// TIA Portal V17 export
// export: Created 2023-02-14T02:49:39.5432232Z, ExportSetting WithDefaults, DisplayName Totally Integrated Automation Portal, DisplayVersion V17, DisplayName TIA Portal Openness, DisplayVersion V17, DisplayName TIA Portal Teamcenter Gateway, DisplayVersion V17, DisplayName TIA Portal Version Control Interface, DisplayVersion V17, DisplayName SINAMICS Startdrive Advanced, DisplayVersion V17, DisplayName SINAMICS Startdrive G130, G150, S120, S150, SINAMICS MV, S210, DisplayVersion V17, DisplayName SINAMICS Startdrive G110M, G120, G120C, G120D, G120P, G115D, DisplayVersion V17, DisplayName STEP 7 Professional, DisplayVersion V17, DisplayName STEP 7 Safety, DisplayVersion V17, DisplayName WinCC Professional, DisplayVersion V17
FUNCTION_BLOCK "BFT_Tomato"   // FB365, LAD
{ S7_Optimized_Access := 'TRUE' }
VERSION : 0.1
// stored: AutoNumber false, IsIECCheckEnabled false, IsRetainMemResEnabled false, MemoryReserve 100, SetENOAutomatically false, UDAEnableTagReadback false
   VAR_INPUT
      IN_FBAV_Inload : Bool;
      IN_FBAV_Outlet : Bool;
      IN_FBAV_Transfer : Bool;
      IN_FBAV_CIP_Tank : Bool;
      IN_FBAV_CIP_Line : Bool;
      IN_FBAV_Vinegar : Bool;
      IN_FBAV_ProWater : Bool;
      IN_FBP_Inload : Bool;
      IN_FBP_Inload_SP : Real;
      IN_FBP_Transfer : Bool;
      IN_FBP_Transfer_SP : Real;
      IN_FBP_CIP : Bool;
      IN_FBP_CIP_Sp : Real;
      IN_LT01 : Real;
      "LCS Start" : Bool;
      "LCS Stop" : Bool;
      "LCS EMS" : Bool;
      IN_Dose_Run : Bool;
      IN_Dose_Held : Bool;
      IN_Dose_Complete : Bool;
      IN_Dose_Header_1 : Bool;
      IN_Dose_Header_2 : Bool;
      IN_Dose_Valve_Cmd : Bool;
      IN_Dose_Pump_Cmd : Bool;
      IN_Dose_Pump_Sp : Real;
      IN_Dose_LineOK : Bool;
      "Inload Busy" : Bool;
      "CIP Pulse" : Bool;
      "CIP Supply ON" : Bool;
      "CIP Req OK" : Bool;
      "CIP Complete" : Bool;
      "CIP Busy" : Bool;
      "Vinegar Available" : Bool;
      "Vinegar Tank Ready" : Bool;
      "Vinegar Prod Ready" : Bool;
      "Vinegar Valve Open" : Bool;
      "Vinegar Pump Run" : Bool;
      IN_FT_Vinegar : Real;
      ProWater_Req_OK : Bool;
      IN_LDT : Date_And_Time;
   END_VAR
   VAR_OUTPUT
      Out_AV_Inload : Bool;
      Out_AV_Outlet : Bool;
      Out_AV_Transfer : Bool;
      Out_AV_CIP_Tank : Bool;
      Out_AV_CIP_Line : Bool;
      Out_AV_Vinegar : Bool;
      Out_AV_ProWater : Bool;
      Out_P_Inload : Bool;
      Out_P_Inload_Sp : Real;
      Out_P_Transfer : Bool;
      Out_P_Transfer_Sp : Real;
      Out_P_CIP : Bool;
      Out_P_CIP_Sp : Real;
      Out_XA : Bool;
      Out_XA_Speed : Real;
      "Vinegar Req" : Bool;
      ProWater_Req : Bool;
      Out_CIP_Req : Bool;
      Out_CIP_LineOpen : Bool;
   END_VAR
   VAR
      Cmd : Struct
         Inload_Tomato : Bool;
         Inload_ProWater : Bool;
         Ready_for_Tranfer : Bool;
         CIP_Tank : Bool;
         CIP_Line : Bool;
         Agitator_SpeedMode : Bool;
         Agitator_Mode : Bool;
         Agitator_Man_OnOff : Bool;
      END_STRUCT;
   END_VAR
   VAR RETAIN
      Param : Struct
         SP_Level_LL : Real := 10.0;
         SP_Level_ML : Real := 80.0;
         SP_Level_HL : Real := 100.0;
         SP_Level_Agi_ON1 : Real := 20.0;
         SP_Level_Agi_OFF1 : Real := 60.0;
         SP_Level_Agi_ON2 : Real := 62.0;
         SP_Level_Agi_OFF2 : Real := 80.0;
         SP_Level_Agi_ON3 : Real := 82.0;
         Agitator_SP_Speed : Real := 50.0;
         SupplyPump_SP_Speed : Real := 80.0;
         L_Hi_Lim : Real := 100.0;
         L_Lo_Lim : Real := 0.0;
         L_Hys : Real := 2.0;
         FlushingTime : DInt := 10000;
         CIP_Trf_SP_Speed : Real := 80.0;
         CIP_Ret_ON_SP : Real := 5.0;
         CIP_Ret_OFF_SP : Real;
      END_STRUCT;
   END_VAR
   VAR
      State : Struct   // Tank in loading state
         Tank_LL : Bool;
         Tank_ML : Bool;
         Tank_HL : Bool;
         Tank_inCIP : Bool;
         Tank_CIP_Enable : Bool;
         Line_inCIP : Bool;
         Line_CIP_Enable : Bool;
         CIP_Return_On : Bool;
         Inloading : Bool;
         Inload_Enable : Bool;
         Ready_For_Transfer : Bool;
         Ready_For_Transfer_Ena : Bool;
         Tank_Available : Bool;
         Transfer_On_Prog : Bool;
         L_Agi_ON1 : Bool;
         L_Agi_ON2 : Bool;
         L_Agi_ON3 : Bool;
         "Dose EN" : Bool;
         Inloading_ProWater : Bool;
         Inloading_Tomato : Bool;
      END_STRUCT;
      Dose : Struct
         Dose_Start : DWord;
         Dose_Pause : DWord;
         Dose_Stop : DWord;
         Dose_State : DWord;
      END_STRUCT;
      alwaysON : Bool;
      L_Hys_Abs : Real;
      Hys_Level_HL : Real;
      Hys_Level_ML : Real;
      Hys_Level_LL : Real;
      Hys_Level_Agi : Real;
      r : Struct
         PosE1 : Bool;
         PosE2 : Bool;
         PosE3 : Bool;
         PosE4 : Bool;
         PosE5 : Bool;
         PosE6 : Bool;
         PosE7 : Bool;
         PosE8 : Bool;
         PosE9 : Bool;
         PosE10 : Bool;
         PosE11 : Bool;
         PosE12 : Bool;
         PosE13 : Bool;
         PosE14 : Bool;
         PosE15 : Bool;
         PosE16 : Bool;
         PosE17 : Bool;
         PosE18 : Bool;
         PosE19 : Bool;
         PosE20 : Bool;
         PosE21 : Bool;
         PosE22 : Bool;
         PosE23 : Bool;
         PosE24 : Bool;
         PosE25 : Bool;
         PosE26 : Bool;
         PosE27 : Bool;
         PosE28 : Bool;
         PosE29 : Bool;
         PosE30 : Bool;
         PosE31 : Bool;
         PosE32 : Bool;
      END_STRUCT;
      Actuator : Struct
         AV_Inload_Tomato : Bool;
         AV_Inload_ProWater : Bool;
         AV_Outlet : Bool;
         AV_Transfer : Bool;
         AV_CIP_Tank : Bool;
         AV_CIP_Line : Bool;
         P_Transfer : Bool;
         P_Inload : Bool;
         P_CIP : Bool;
         Agitator_level : Bool;
         LCS_OnOff : Bool;
      END_STRUCT;
      FlushingTim : TON_TIME;
      SPumpTim { S7_SetPoint := 'True'} : TON_TIME;
      AVinloadTim { S7_SetPoint := 'True'} : TON_TIME;
      L_AgiTim { S7_SetPoint := 'True'} : TON_TIME;
      SP_Vinegar { S7_SetPoint := 'True'} : "RawDose";
      Dose_Vinegar { S7_SetPoint := 'True'} : "DOSE";
      Vinegar_Ready_State { S7_SetPoint := 'True'} : Bool;
      Vinegar_EN : Bool;
      Pump_TF_On_Time { S7_SetPoint := 'True'} : TON_TIME;
   END_VAR
   VAR_TEMP   // added for the SCL form of the ladder/FBD networks
      _w1 : Bool;
      _w2 : Bool;
   END_VAR
BEGIN

REGION Network 1: Always_ON
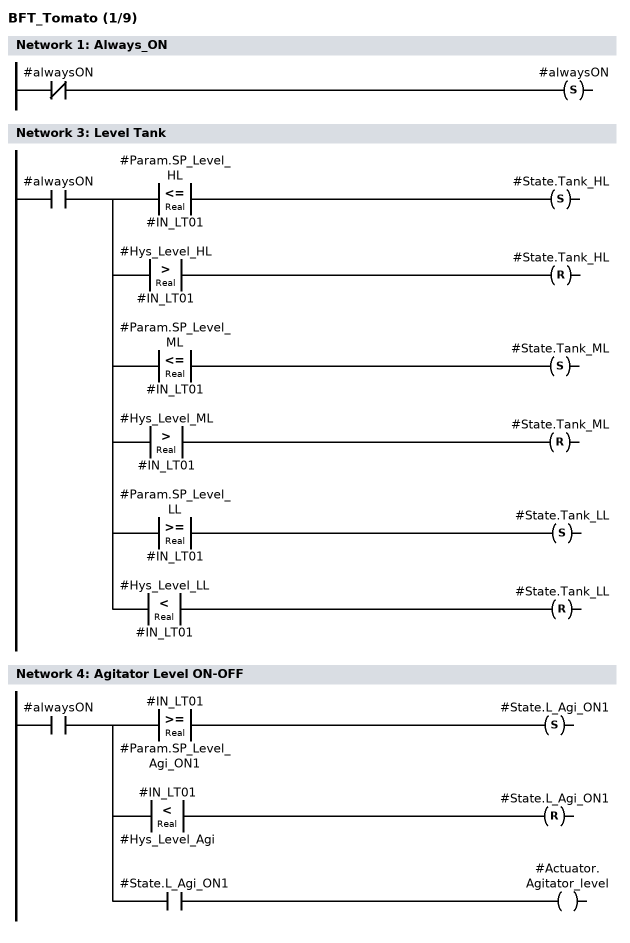
   RUNG wire#powerrail
      I_Contact( #alwaysON )
      S_Coil( #alwaysON )
   END_RUNG
   // the same network as SCL:
   IF NOT #alwaysON THEN #alwaysON := TRUE; END_IF;
END_REGION

NETWORK
TITLE = Hys Calculation
//Level Hys Absolute
      L     #Param.L_Hi_Lim;
      L     #Param.L_Lo_Lim;
      -R;
      L     100.0;
      /R;
      L     #Param.L_Hys;
      *R;
      T     #L_Hys_Abs;
//Tank High Level
      L     #Param.SP_Level_HL;
      L     #L_Hys_Abs;
      -R;
      T     #Hys_Level_HL;
//Tank Mid Level
      L     #Param.SP_Level_ML;
      L     #L_Hys_Abs;
      -R;
      T     #Hys_Level_ML;
//Tank Low Level
      L     #Param.SP_Level_LL;
      L     #L_Hys_Abs;
      +R;
      T     #Hys_Level_LL;
//Level Agi
      L     #Param.SP_Level_Agi_ON1;
      L     #L_Hys_Abs;
      -R;
      T     #Hys_Level_Agi;



REGION Network 3: Level Tank
   RUNG wire#powerrail
      Contact( #alwaysON )
      wire#w1
      { S7_Templates := "SrcType := Real" } LE_Contact(in1 := #Param.SP_Level_HL, in2 := #IN_LT01)
      S_Coil( #State.Tank_HL )
   END_RUNG
   RUNG wire#w1
      { S7_Templates := "SrcType := Real" } GT_Contact(in1 := #Hys_Level_HL, in2 := #IN_LT01)
      R_Coil( #State.Tank_HL )
   END_RUNG
   RUNG wire#w1
      { S7_Templates := "SrcType := Real" } LE_Contact(in1 := #Param.SP_Level_ML, in2 := #IN_LT01)
      S_Coil( #State.Tank_ML )
   END_RUNG
   RUNG wire#w1
      { S7_Templates := "SrcType := Real" } GT_Contact(in1 := #Hys_Level_ML, in2 := #IN_LT01)
      R_Coil( #State.Tank_ML )
   END_RUNG
   RUNG wire#w1
      { S7_Templates := "SrcType := Real" } GE_Contact(in1 := #Param.SP_Level_LL, in2 := #IN_LT01)
      S_Coil( #State.Tank_LL )
   END_RUNG
   RUNG wire#w1
      { S7_Templates := "SrcType := Real" } LT_Contact(in1 := #Hys_Level_LL, in2 := #IN_LT01)
      R_Coil( #State.Tank_LL )
   END_RUNG
   // the same network as SCL:
   IF #alwaysON AND (#Param.SP_Level_HL <= #IN_LT01) THEN #State.Tank_HL := TRUE; END_IF;
   IF #alwaysON AND (#Hys_Level_HL > #IN_LT01) THEN #State.Tank_HL := FALSE; END_IF;
   IF #alwaysON AND (#Param.SP_Level_ML <= #IN_LT01) THEN #State.Tank_ML := TRUE; END_IF;
   IF #alwaysON AND (#Hys_Level_ML > #IN_LT01) THEN #State.Tank_ML := FALSE; END_IF;
   IF #alwaysON AND (#Param.SP_Level_LL >= #IN_LT01) THEN #State.Tank_LL := TRUE; END_IF;
   IF #alwaysON AND (#Hys_Level_LL < #IN_LT01) THEN #State.Tank_LL := FALSE; END_IF;
END_REGION

REGION Network 4: Agitator Level ON-OFF
   RUNG wire#powerrail
      Contact( #alwaysON )
      wire#w1
      { S7_Templates := "SrcType := Real" } GE_Contact(in1 := #IN_LT01, in2 := #Param.SP_Level_Agi_ON1)
      S_Coil( #State.L_Agi_ON1 )
   END_RUNG
   RUNG wire#w1
      { S7_Templates := "SrcType := Real" } LT_Contact(in1 := #IN_LT01, in2 := #Hys_Level_Agi)
      R_Coil( #State.L_Agi_ON1 )
   END_RUNG
   RUNG wire#w1
      Contact( #State.L_Agi_ON1 )
      Coil( #Actuator.Agitator_level )
   END_RUNG
   // the same network as SCL:
   IF #alwaysON AND (#IN_LT01 >= #Param.SP_Level_Agi_ON1) THEN #State.L_Agi_ON1 := TRUE; END_IF;
   IF #alwaysON AND (#IN_LT01 < #Hys_Level_Agi) THEN #State.L_Agi_ON1 := FALSE; END_IF;
   #Actuator.Agitator_level := #alwaysON AND #State.L_Agi_ON1;
END_REGION

REGION Network 5: Agitator
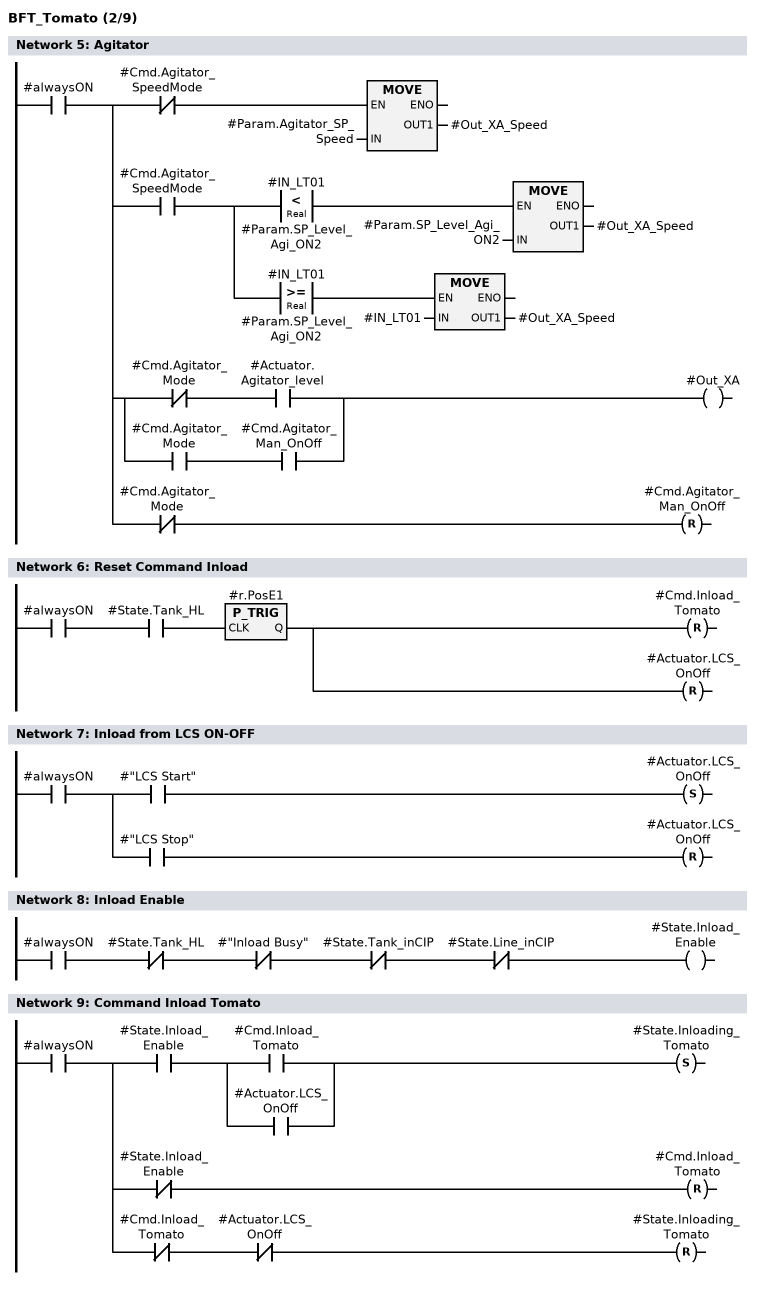
   RUNG wire#powerrail
      Contact( #alwaysON )
      wire#w1
      I_Contact( #Cmd.Agitator_SpeedMode )
      Move(in := #Param.Agitator_SP_Speed, out1 => #Out_XA_Speed)
   END_RUNG
   RUNG wire#w1
      Contact( #Cmd.Agitator_SpeedMode )
      wire#w2
      { S7_Templates := "SrcType := Real" } LT_Contact(in1 := #IN_LT01, in2 := #Param.SP_Level_Agi_ON2)
      Move(in := #Param.SP_Level_Agi_ON2, out1 => #Out_XA_Speed)
   END_RUNG
   RUNG wire#w2
      { S7_Templates := "SrcType := Real" } GE_Contact(in1 := #IN_LT01, in2 := #Param.SP_Level_Agi_ON2)
      Move(in := #IN_LT01, out1 => #Out_XA_Speed)
   END_RUNG
   RUNG wire#w1
      I_Contact( #Cmd.Agitator_Mode )
      Contact( #Actuator.Agitator_level )
      wire#w3
      Coil( #Out_XA )
   END_RUNG
   RUNG wire#w1
      Contact( #Cmd.Agitator_Mode )
      Contact( #Cmd.Agitator_Man_OnOff )
   END_RUNG wire#w3
   RUNG wire#w1
      I_Contact( #Cmd.Agitator_Mode )
      R_Coil( #Cmd.Agitator_Man_OnOff )
   END_RUNG
   // the same network as SCL:
   IF #alwaysON AND NOT #Cmd.Agitator_SpeedMode THEN #Out_XA_Speed := #Param.Agitator_SP_Speed; END_IF;
   #_w1 := #alwaysON AND #Cmd.Agitator_SpeedMode;
   IF #_w1 AND (#IN_LT01 < #Param.SP_Level_Agi_ON2) THEN #Out_XA_Speed := #Param.SP_Level_Agi_ON2; END_IF;
   IF #_w1 AND (#IN_LT01 >= #Param.SP_Level_Agi_ON2) THEN #Out_XA_Speed := #IN_LT01; END_IF;
   #Out_XA := #alwaysON AND ((NOT #Cmd.Agitator_Mode AND #Actuator.Agitator_level) OR (#Cmd.Agitator_Mode AND #Cmd.Agitator_Man_OnOff));
   IF #alwaysON AND NOT #Cmd.Agitator_Mode THEN #Cmd.Agitator_Man_OnOff := FALSE; END_IF;
END_REGION

REGION Network 6: Reset Command Inload
   RUNG wire#powerrail
      Contact( #alwaysON )
      Contact( #State.Tank_HL )
      P_Trig( #r.PosE1 )
      wire#w1
      R_Coil( #Cmd.Inload_Tomato )
   END_RUNG
   RUNG wire#w1
      R_Coil( #Actuator.LCS_OnOff )
   END_RUNG
   // the same network as SCL:
   #_w1 := #alwaysON AND #State.Tank_HL;
   #_w2 := #_w1 AND NOT #r.PosE1;   // rising edge
   #r.PosE1 := #_w1;
   IF #_w2 THEN
       #Cmd.Inload_Tomato := FALSE;
       #Actuator.LCS_OnOff := FALSE;
   END_IF;
END_REGION

REGION Network 7: Inload from LCS ON-OFF
   RUNG wire#powerrail
      Contact( #alwaysON )
      wire#w1
      Contact( #"LCS Start" )
      S_Coil( #Actuator.LCS_OnOff )
   END_RUNG
   RUNG wire#w1
      Contact( #"LCS Stop" )
      R_Coil( #Actuator.LCS_OnOff )
   END_RUNG
   // the same network as SCL:
   IF #alwaysON AND #"LCS Start" THEN #Actuator.LCS_OnOff := TRUE; END_IF;
   IF #alwaysON AND #"LCS Stop" THEN #Actuator.LCS_OnOff := FALSE; END_IF;
END_REGION

REGION Network 8: Inload Enable
   RUNG wire#powerrail
      Contact( #alwaysON )
      I_Contact( #State.Tank_HL )
      I_Contact( #"Inload Busy" )
      I_Contact( #State.Tank_inCIP )
      I_Contact( #State.Line_inCIP )
      Coil( #State.Inload_Enable )
   END_RUNG
   // the same network as SCL:
   #State.Inload_Enable := #alwaysON AND NOT #State.Tank_HL AND NOT #"Inload Busy" AND NOT #State.Tank_inCIP AND NOT #State.Line_inCIP;
END_REGION

REGION Network 9: Command Inload Tomato
   RUNG wire#powerrail
      Contact( #alwaysON )
      wire#w1
      Contact( #State.Inload_Enable )
      wire#w2
      Contact( #Cmd.Inload_Tomato )
      wire#w3
      S_Coil( #State.Inloading_Tomato )
   END_RUNG
   RUNG wire#w2
      Contact( #Actuator.LCS_OnOff )
   END_RUNG wire#w3
   RUNG wire#w1
      I_Contact( #State.Inload_Enable )
      R_Coil( #Cmd.Inload_Tomato )
   END_RUNG
   RUNG wire#w1
      I_Contact( #Cmd.Inload_Tomato )
      I_Contact( #Actuator.LCS_OnOff )
      R_Coil( #State.Inloading_Tomato )
   END_RUNG
   // the same network as SCL:
   IF #alwaysON AND #State.Inload_Enable AND (#Cmd.Inload_Tomato OR #Actuator.LCS_OnOff) THEN
       #State.Inloading_Tomato := TRUE;
   END_IF;
   IF #alwaysON AND NOT #State.Inload_Enable THEN #Cmd.Inload_Tomato := FALSE; END_IF;
   IF #alwaysON AND NOT #Cmd.Inload_Tomato AND NOT #Actuator.LCS_OnOff THEN
       #State.Inloading_Tomato := FALSE;
   END_IF;
END_REGION

REGION Network 10: Command Inload Process Water
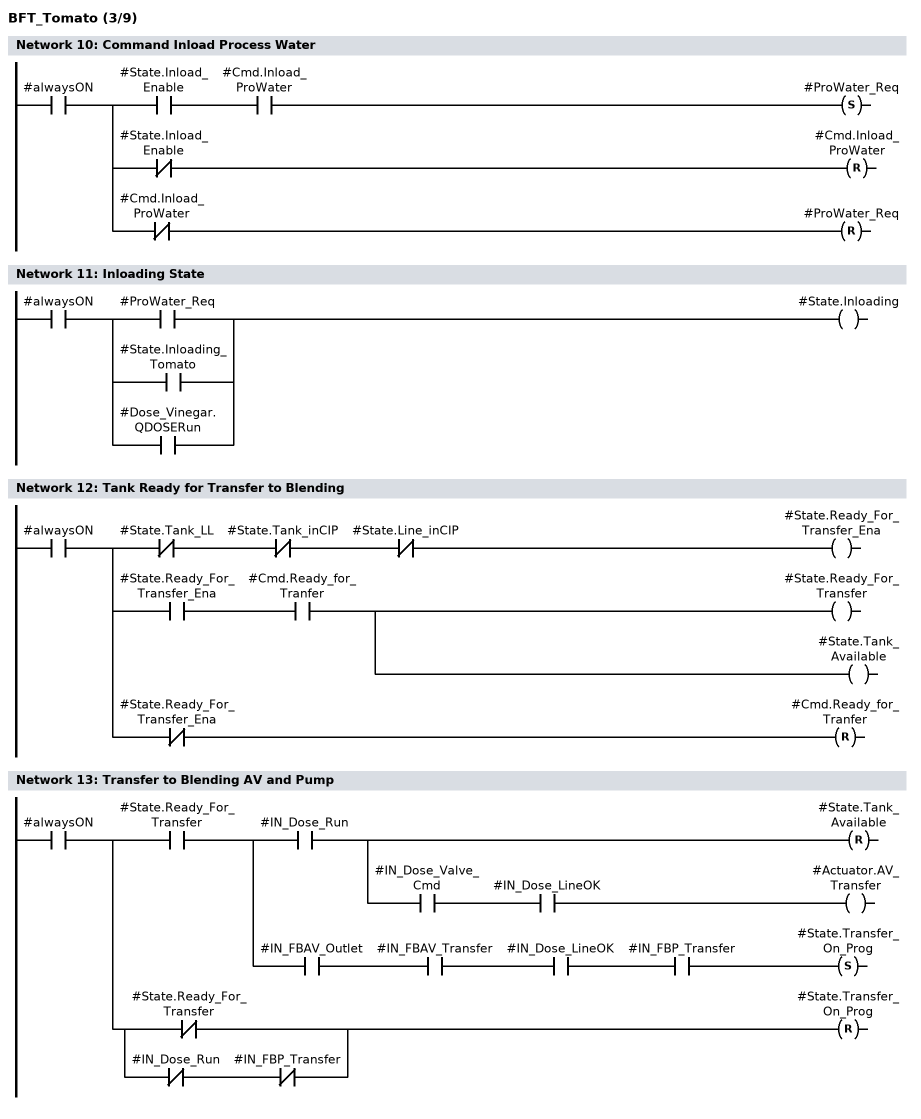
   RUNG wire#powerrail
      Contact( #alwaysON )
      wire#w1
      Contact( #State.Inload_Enable )
      Contact( #Cmd.Inload_ProWater )
      S_Coil( #ProWater_Req )
   END_RUNG
   RUNG wire#w1
      I_Contact( #State.Inload_Enable )
      R_Coil( #Cmd.Inload_ProWater )
   END_RUNG
   RUNG wire#w1
      I_Contact( #Cmd.Inload_ProWater )
      R_Coil( #ProWater_Req )
   END_RUNG
   // the same network as SCL:
   IF #alwaysON AND #State.Inload_Enable AND #Cmd.Inload_ProWater THEN #ProWater_Req := TRUE; END_IF;
   IF #alwaysON AND NOT #State.Inload_Enable THEN #Cmd.Inload_ProWater := FALSE; END_IF;
   IF #alwaysON AND NOT #Cmd.Inload_ProWater THEN #ProWater_Req := FALSE; END_IF;
END_REGION

REGION Network 11: Inloading State
   RUNG wire#powerrail
      Contact( #alwaysON )
      wire#w1
      Contact( #ProWater_Req )
      wire#w2
      Coil( #State.Inloading )
   END_RUNG
   RUNG wire#w1
      Contact( #State.Inloading_Tomato )
   END_RUNG wire#w2
   RUNG wire#w1
      Contact( #Dose_Vinegar.QDOSERun )
   END_RUNG wire#w2
   // the same network as SCL:
   #State.Inloading := #alwaysON AND (#ProWater_Req OR #State.Inloading_Tomato OR #Dose_Vinegar.QDOSERun);
END_REGION

REGION Network 12: Tank Ready for Transfer to Blending
   RUNG wire#powerrail
      Contact( #alwaysON )
      wire#w1
      I_Contact( #State.Tank_LL )
      I_Contact( #State.Tank_inCIP )
      I_Contact( #State.Line_inCIP )
      Coil( #State.Ready_For_Transfer_Ena )
   END_RUNG
   RUNG wire#w1
      Contact( #State.Ready_For_Transfer_Ena )
      Contact( #Cmd.Ready_for_Tranfer )
      wire#w2
      Coil( #State.Ready_For_Transfer )
   END_RUNG
   RUNG wire#w2
      Coil( #State.Tank_Available )
   END_RUNG
   RUNG wire#w1
      I_Contact( #State.Ready_For_Transfer_Ena )
      R_Coil( #Cmd.Ready_for_Tranfer )
   END_RUNG
   // the same network as SCL:
   #State.Ready_For_Transfer_Ena := #alwaysON AND NOT #State.Tank_LL AND NOT #State.Tank_inCIP AND NOT #State.Line_inCIP;
   #State.Ready_For_Transfer := #alwaysON AND #State.Ready_For_Transfer_Ena AND #Cmd.Ready_for_Tranfer;
   #State.Tank_Available := #State.Ready_For_Transfer;
   IF #alwaysON AND NOT #State.Ready_For_Transfer_Ena THEN #Cmd.Ready_for_Tranfer := FALSE; END_IF;
END_REGION

REGION Network 13: Transfer to Blending AV and Pump
   RUNG wire#powerrail
      Contact( #alwaysON )
      wire#w1
      Contact( #State.Ready_For_Transfer )
      wire#w2
      Contact( #IN_Dose_Run )
      wire#w3
      R_Coil( #State.Tank_Available )
   END_RUNG
   RUNG wire#w3
      Contact( #IN_Dose_Valve_Cmd )
      Contact( #IN_Dose_LineOK )
      Coil( #Actuator.AV_Transfer )
   END_RUNG
   RUNG wire#w2
      Contact( #IN_FBAV_Outlet )
      Contact( #IN_FBAV_Transfer )
      Contact( #IN_Dose_LineOK )
      Contact( #IN_FBP_Transfer )
      S_Coil( #State.Transfer_On_Prog )
   END_RUNG
   RUNG wire#w1
      I_Contact( #State.Ready_For_Transfer )
      wire#w4
      R_Coil( #State.Transfer_On_Prog )
   END_RUNG
   RUNG wire#w1
      I_Contact( #IN_Dose_Run )
      I_Contact( #IN_FBP_Transfer )
   END_RUNG wire#w4
   // the same network as SCL:
   #_w1 := #alwaysON AND #State.Ready_For_Transfer;
   #_w2 := #_w1 AND #IN_Dose_Run;
   IF #_w2 THEN #State.Tank_Available := FALSE; END_IF;
   #Actuator.AV_Transfer := #_w2 AND #IN_Dose_Valve_Cmd AND #IN_Dose_LineOK;
   IF #_w1 AND #IN_FBAV_Outlet AND #IN_FBAV_Transfer AND #IN_Dose_LineOK AND #IN_FBP_Transfer THEN
       #State.Transfer_On_Prog := TRUE;
   END_IF;
   IF #alwaysON AND (NOT #State.Ready_For_Transfer OR (NOT #IN_Dose_Run AND NOT #IN_FBP_Transfer)) THEN
       #State.Transfer_On_Prog := FALSE;
   END_IF;
END_REGION

REGION Network 14: Command CIP
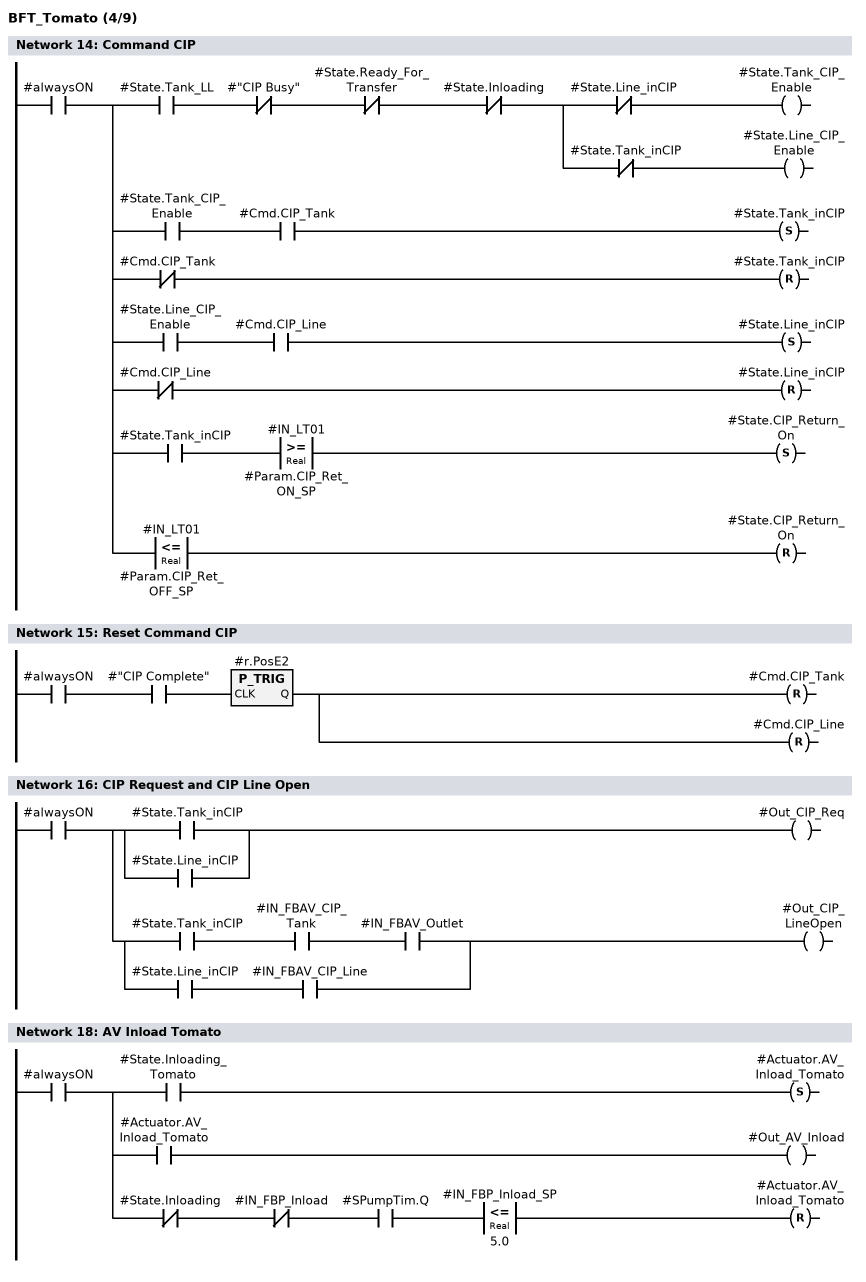
   RUNG wire#powerrail
      Contact( #alwaysON )
      wire#w1
      Contact( #State.Tank_LL )
      I_Contact( #"CIP Busy" )
      I_Contact( #State.Ready_For_Transfer )
      I_Contact( #State.Inloading )
      wire#w2
      I_Contact( #State.Line_inCIP )
      Coil( #State.Tank_CIP_Enable )
   END_RUNG
   RUNG wire#w2
      I_Contact( #State.Tank_inCIP )
      Coil( #State.Line_CIP_Enable )
   END_RUNG
   RUNG wire#w1
      Contact( #State.Tank_CIP_Enable )
      Contact( #Cmd.CIP_Tank )
      S_Coil( #State.Tank_inCIP )
   END_RUNG
   RUNG wire#w1
      I_Contact( #Cmd.CIP_Tank )
      R_Coil( #State.Tank_inCIP )
   END_RUNG
   RUNG wire#w1
      Contact( #State.Line_CIP_Enable )
      Contact( #Cmd.CIP_Line )
      S_Coil( #State.Line_inCIP )
   END_RUNG
   RUNG wire#w1
      I_Contact( #Cmd.CIP_Line )
      R_Coil( #State.Line_inCIP )
   END_RUNG
   RUNG wire#w1
      Contact( #State.Tank_inCIP )
      { S7_Templates := "SrcType := Real" } GE_Contact(in1 := #IN_LT01, in2 := #Param.CIP_Ret_ON_SP)
      S_Coil( #State.CIP_Return_On )
   END_RUNG
   RUNG wire#w1
      { S7_Templates := "SrcType := Real" } LE_Contact(in1 := #IN_LT01, in2 := #Param.CIP_Ret_OFF_SP)
      R_Coil( #State.CIP_Return_On )
   END_RUNG
   // the same network as SCL:
   #_w1 := #alwaysON AND #State.Tank_LL AND NOT #"CIP Busy" AND NOT #State.Ready_For_Transfer AND NOT #State.Inloading;
   #State.Tank_CIP_Enable := #_w1 AND NOT #State.Line_inCIP;
   #State.Line_CIP_Enable := #_w1 AND NOT #State.Tank_inCIP;
   IF #alwaysON AND #State.Tank_CIP_Enable AND #Cmd.CIP_Tank THEN #State.Tank_inCIP := TRUE; END_IF;
   IF #alwaysON AND NOT #Cmd.CIP_Tank THEN #State.Tank_inCIP := FALSE; END_IF;
   IF #alwaysON AND #State.Line_CIP_Enable AND #Cmd.CIP_Line THEN #State.Line_inCIP := TRUE; END_IF;
   IF #alwaysON AND NOT #Cmd.CIP_Line THEN #State.Line_inCIP := FALSE; END_IF;
   IF #alwaysON AND #State.Tank_inCIP AND (#IN_LT01 >= #Param.CIP_Ret_ON_SP) THEN
       #State.CIP_Return_On := TRUE;
   END_IF;
   IF #alwaysON AND (#IN_LT01 <= #Param.CIP_Ret_OFF_SP) THEN #State.CIP_Return_On := FALSE; END_IF;
END_REGION

REGION Network 15: Reset Command CIP
   RUNG wire#powerrail
      Contact( #alwaysON )
      Contact( #"CIP Complete" )
      P_Trig( #r.PosE2 )
      wire#w1
      R_Coil( #Cmd.CIP_Tank )
   END_RUNG
   RUNG wire#w1
      R_Coil( #Cmd.CIP_Line )
   END_RUNG
   // the same network as SCL:
   #_w1 := #alwaysON AND #"CIP Complete";
   #_w2 := #_w1 AND NOT #r.PosE2;   // rising edge
   #r.PosE2 := #_w1;
   IF #_w2 THEN
       #Cmd.CIP_Tank := FALSE;
       #Cmd.CIP_Line := FALSE;
   END_IF;
END_REGION

REGION Network 16: CIP Request and CIP Line Open
   RUNG wire#powerrail
      Contact( #alwaysON )
      wire#w1
      Contact( #State.Tank_inCIP )
      wire#w2
      Coil( #Out_CIP_Req )
   END_RUNG
   RUNG wire#w1
      Contact( #State.Line_inCIP )
   END_RUNG wire#w2
   RUNG wire#w1
      Contact( #State.Tank_inCIP )
      Contact( #IN_FBAV_CIP_Tank )
      Contact( #IN_FBAV_Outlet )
      wire#w3
      Coil( #Out_CIP_LineOpen )
   END_RUNG
   RUNG wire#w1
      Contact( #State.Line_inCIP )
      Contact( #IN_FBAV_CIP_Line )
   END_RUNG wire#w3
   // the same network as SCL:
   #Out_CIP_Req := #alwaysON AND (#State.Tank_inCIP OR #State.Line_inCIP);
   #Out_CIP_LineOpen := #alwaysON AND ((#State.Tank_inCIP AND #IN_FBAV_CIP_Tank AND #IN_FBAV_Outlet) OR (#State.Line_inCIP AND #IN_FBAV_CIP_Line));
END_REGION

REGION Network 18: AV Inload Tomato
   RUNG wire#powerrail
      Contact( #alwaysON )
      wire#w1
      Contact( #State.Inloading_Tomato )
      S_Coil( #Actuator.AV_Inload_Tomato )
   END_RUNG
   RUNG wire#w1
      Contact( #Actuator.AV_Inload_Tomato )
      Coil( #Out_AV_Inload )
   END_RUNG
   RUNG wire#w1
      I_Contact( #State.Inloading )
      I_Contact( #IN_FBP_Inload )
      Contact( #SPumpTim.Q )
      { S7_Templates := "SrcType := Real" } LE_Contact(in1 := #IN_FBP_Inload_SP, in2 := 5.0)
      R_Coil( #Actuator.AV_Inload_Tomato )
   END_RUNG
   // the same network as SCL:
   IF #alwaysON AND #State.Inloading_Tomato THEN #Actuator.AV_Inload_Tomato := TRUE; END_IF;
   #Out_AV_Inload := #alwaysON AND #Actuator.AV_Inload_Tomato;
   IF #alwaysON AND NOT #State.Inloading AND NOT #IN_FBP_Inload AND #SPumpTim.Q AND (#IN_FBP_Inload_SP <= 5.0) THEN
       #Actuator.AV_Inload_Tomato := FALSE;
   END_IF;
END_REGION

REGION Network 19: AV Inload ProWater
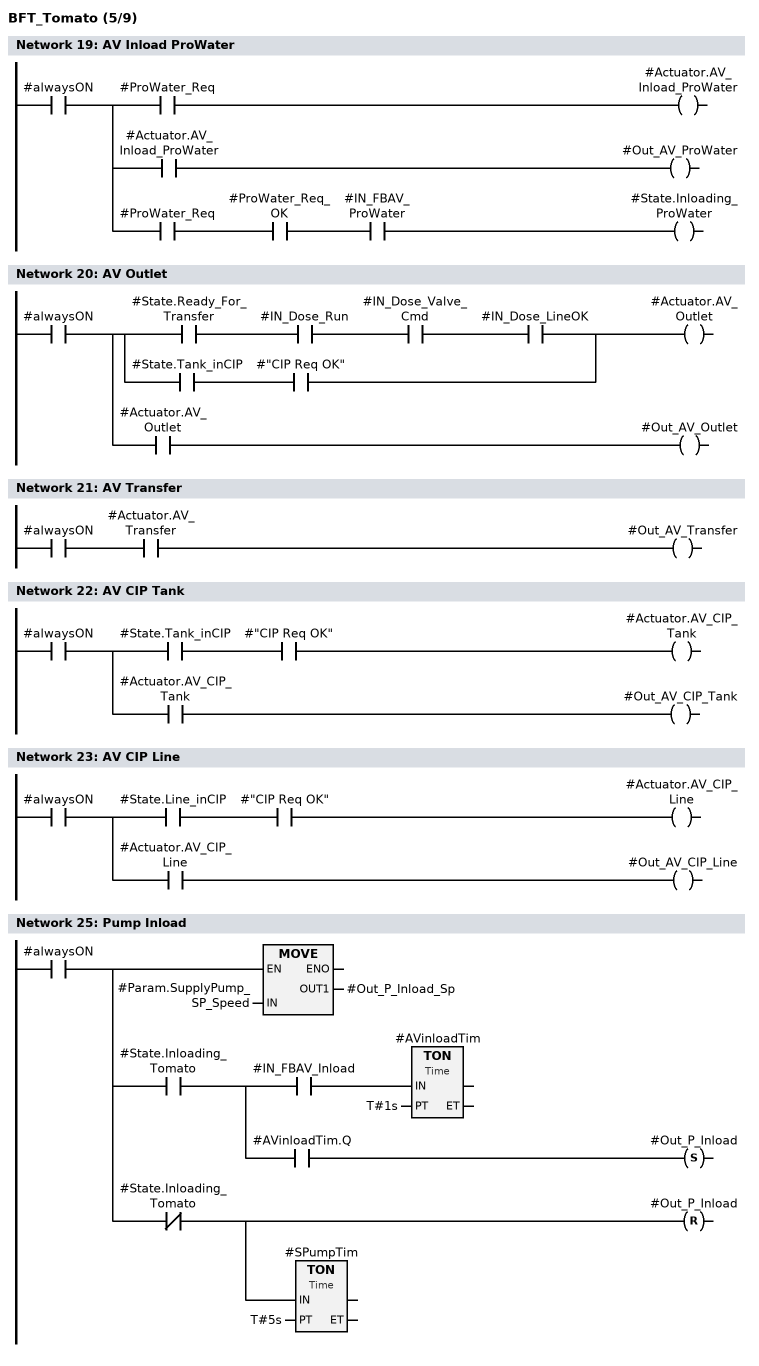
   RUNG wire#powerrail
      Contact( #alwaysON )
      wire#w1
      Contact( #ProWater_Req )
      Coil( #Actuator.AV_Inload_ProWater )
   END_RUNG
   RUNG wire#w1
      Contact( #Actuator.AV_Inload_ProWater )
      Coil( #Out_AV_ProWater )
   END_RUNG
   RUNG wire#w1
      Contact( #ProWater_Req )
      Contact( #ProWater_Req_OK )
      Contact( #IN_FBAV_ProWater )
      Coil( #State.Inloading_ProWater )
   END_RUNG
   // the same network as SCL:
   #Actuator.AV_Inload_ProWater := #alwaysON AND #ProWater_Req;
   #Out_AV_ProWater := #alwaysON AND #Actuator.AV_Inload_ProWater;
   #State.Inloading_ProWater := #alwaysON AND #ProWater_Req AND #ProWater_Req_OK AND #IN_FBAV_ProWater;
END_REGION

REGION Network 20: AV Outlet
   RUNG wire#powerrail
      Contact( #alwaysON )
      wire#w1
      Contact( #State.Ready_For_Transfer )
      Contact( #IN_Dose_Run )
      Contact( #IN_Dose_Valve_Cmd )
      Contact( #IN_Dose_LineOK )
      wire#w2
      Coil( #Actuator.AV_Outlet )
   END_RUNG
   RUNG wire#w1
      Contact( #State.Tank_inCIP )
      Contact( #"CIP Req OK" )
   END_RUNG wire#w2
   RUNG wire#w1
      Contact( #Actuator.AV_Outlet )
      Coil( #Out_AV_Outlet )
   END_RUNG
   // the same network as SCL:
   #Actuator.AV_Outlet := #alwaysON AND ((#State.Ready_For_Transfer AND #IN_Dose_Run AND #IN_Dose_Valve_Cmd AND #IN_Dose_LineOK) OR (#State.Tank_inCIP AND #"CIP Req OK"));
   #Out_AV_Outlet := #alwaysON AND #Actuator.AV_Outlet;
END_REGION

REGION Network 21: AV Transfer
   RUNG wire#powerrail
      Contact( #alwaysON )
      Contact( #Actuator.AV_Transfer )
      Coil( #Out_AV_Transfer )
   END_RUNG
   // the same network as SCL:
   #Out_AV_Transfer := #alwaysON AND #Actuator.AV_Transfer;
END_REGION

REGION Network 22: AV CIP Tank
   RUNG wire#powerrail
      Contact( #alwaysON )
      wire#w1
      Contact( #State.Tank_inCIP )
      Contact( #"CIP Req OK" )
      Coil( #Actuator.AV_CIP_Tank )
   END_RUNG
   RUNG wire#w1
      Contact( #Actuator.AV_CIP_Tank )
      Coil( #Out_AV_CIP_Tank )
   END_RUNG
   // the same network as SCL:
   #Actuator.AV_CIP_Tank := #alwaysON AND #State.Tank_inCIP AND #"CIP Req OK";
   #Out_AV_CIP_Tank := #alwaysON AND #Actuator.AV_CIP_Tank;
END_REGION

REGION Network 23: AV CIP Line
   RUNG wire#powerrail
      Contact( #alwaysON )
      wire#w1
      Contact( #State.Line_inCIP )
      Contact( #"CIP Req OK" )
      Coil( #Actuator.AV_CIP_Line )
   END_RUNG
   RUNG wire#w1
      Contact( #Actuator.AV_CIP_Line )
      Coil( #Out_AV_CIP_Line )
   END_RUNG
   // the same network as SCL:
   #Actuator.AV_CIP_Line := #alwaysON AND #State.Line_inCIP AND #"CIP Req OK";
   #Out_AV_CIP_Line := #alwaysON AND #Actuator.AV_CIP_Line;
END_REGION

REGION Network 25: Pump Inload
   RUNG wire#powerrail
      Contact( #alwaysON )
      wire#w1
      Move(in := #Param.SupplyPump_SP_Speed, out1 => #Out_P_Inload_Sp)
   END_RUNG
   RUNG wire#w1
      Contact( #State.Inloading_Tomato )
      wire#w2
      Contact( #IN_FBAV_Inload )
      { S7_Templates := "time_type := Time" } #AVinloadTim.TON(pt := T#1s, et =>)
   END_RUNG
   RUNG wire#w2
      Contact( #AVinloadTim.Q )
      S_Coil( #Out_P_Inload )
   END_RUNG
   RUNG wire#w1
      I_Contact( #State.Inloading_Tomato )
      wire#w3
      R_Coil( #Out_P_Inload )
   END_RUNG
   RUNG wire#w3
      { S7_Templates := "time_type := Time" } #SPumpTim.TON(pt := T#5s, et =>)
   END_RUNG
   // the same network as SCL:
   IF #alwaysON THEN #Out_P_Inload_Sp := #Param.SupplyPump_SP_Speed; END_IF;
   #_w1 := #alwaysON AND #State.Inloading_Tomato;
   #AVinloadTim(IN := #_w1 AND #IN_FBAV_Inload, PT := T#1s);   // TON
   IF #_w1 AND #AVinloadTim.Q THEN #Out_P_Inload := TRUE; END_IF;
   #_w2 := #alwaysON AND NOT #State.Inloading_Tomato;
   IF #_w2 THEN #Out_P_Inload := FALSE; END_IF;
   #SPumpTim(IN := #_w2, PT := T#5s);   // TON
END_REGION

REGION Network 26: Pump Transfer
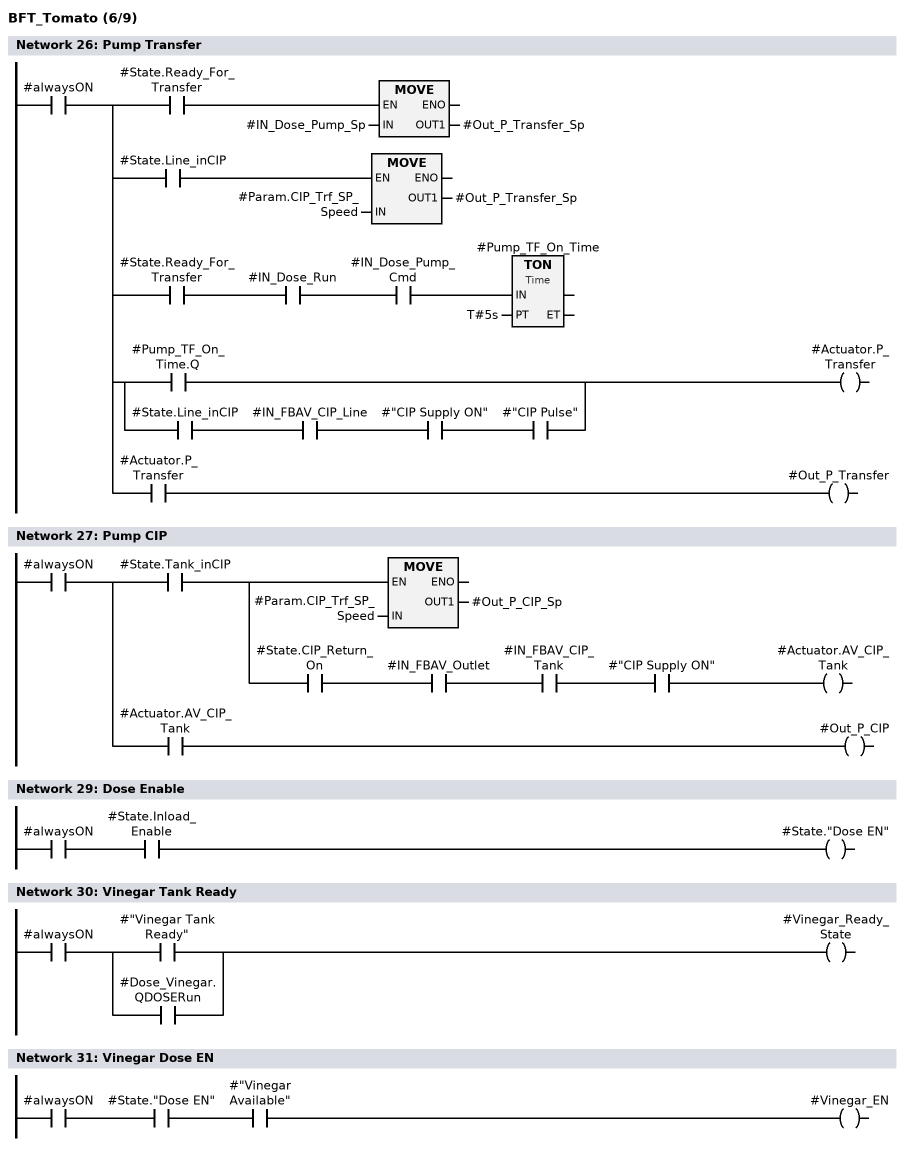
   RUNG wire#powerrail
      Contact( #alwaysON )
      wire#w1
      Contact( #State.Ready_For_Transfer )
      Move(in := #IN_Dose_Pump_Sp, out1 => #Out_P_Transfer_Sp)
   END_RUNG
   RUNG wire#w1
      Contact( #State.Line_inCIP )
      Move(in := #Param.CIP_Trf_SP_Speed, out1 => #Out_P_Transfer_Sp)
   END_RUNG
   RUNG wire#w1
      Contact( #State.Ready_For_Transfer )
      Contact( #IN_Dose_Run )
      Contact( #IN_Dose_Pump_Cmd )
      { S7_Templates := "time_type := Time" } #Pump_TF_On_Time.TON(pt := T#5s, et =>)
   END_RUNG
   RUNG wire#w1
      Contact( #Pump_TF_On_Time.Q )
      wire#w2
      Coil( #Actuator.P_Transfer )
   END_RUNG
   RUNG wire#w1
      Contact( #State.Line_inCIP )
      Contact( #IN_FBAV_CIP_Line )
      Contact( #"CIP Supply ON" )
      Contact( #"CIP Pulse" )
   END_RUNG wire#w2
   RUNG wire#w1
      Contact( #Actuator.P_Transfer )
      Coil( #Out_P_Transfer )
   END_RUNG
   // the same network as SCL:
   IF #alwaysON AND #State.Ready_For_Transfer THEN #Out_P_Transfer_Sp := #IN_Dose_Pump_Sp; END_IF;
   IF #alwaysON AND #State.Line_inCIP THEN #Out_P_Transfer_Sp := #Param.CIP_Trf_SP_Speed; END_IF;
   #Pump_TF_On_Time(IN := #alwaysON AND #State.Ready_For_Transfer AND #IN_Dose_Run AND #IN_Dose_Pump_Cmd,   // TON
                    PT := T#5s);
   #Actuator.P_Transfer := #alwaysON AND (#Pump_TF_On_Time.Q OR (#State.Line_inCIP AND #IN_FBAV_CIP_Line AND #"CIP Supply ON" AND #"CIP Pulse"));
   #Out_P_Transfer := #alwaysON AND #Actuator.P_Transfer;
END_REGION

REGION Network 27: Pump CIP
   RUNG wire#powerrail
      Contact( #alwaysON )
      wire#w1
      Contact( #State.Tank_inCIP )
      wire#w2
      Move(in := #Param.CIP_Trf_SP_Speed, out1 => #Out_P_CIP_Sp)
   END_RUNG
   RUNG wire#w2
      Contact( #State.CIP_Return_On )
      Contact( #IN_FBAV_Outlet )
      Contact( #IN_FBAV_CIP_Tank )
      Contact( #"CIP Supply ON" )
      Coil( #Actuator.AV_CIP_Tank )
   END_RUNG
   RUNG wire#w1
      Contact( #Actuator.AV_CIP_Tank )
      Coil( #Out_P_CIP )
   END_RUNG
   // the same network as SCL:
   #_w1 := #alwaysON AND #State.Tank_inCIP;
   IF #_w1 THEN #Out_P_CIP_Sp := #Param.CIP_Trf_SP_Speed; END_IF;
   #Actuator.AV_CIP_Tank := #_w1 AND #State.CIP_Return_On AND #IN_FBAV_Outlet AND #IN_FBAV_CIP_Tank AND #"CIP Supply ON";
   #Out_P_CIP := #alwaysON AND #Actuator.AV_CIP_Tank;
END_REGION

REGION Network 29: Dose Enable
   RUNG wire#powerrail
      Contact( #alwaysON )
      Contact( #State.Inload_Enable )
      Coil( #State."Dose EN" )
   END_RUNG
   // the same network as SCL:
   #State."Dose EN" := #alwaysON AND #State.Inload_Enable;
END_REGION

REGION Network 30: Vinegar Tank Ready
   RUNG wire#powerrail
      Contact( #alwaysON )
      wire#w1
      Contact( #"Vinegar Tank Ready" )
      wire#w2
      Coil( #Vinegar_Ready_State )
   END_RUNG
   RUNG wire#w1
      Contact( #Dose_Vinegar.QDOSERun )
   END_RUNG wire#w2
   // the same network as SCL:
   #Vinegar_Ready_State := #alwaysON AND (#"Vinegar Tank Ready" OR #Dose_Vinegar.QDOSERun);
END_REGION

REGION Network 31: Vinegar Dose EN
   RUNG wire#powerrail
      Contact( #alwaysON )
      Contact( #State."Dose EN" )
      Contact( #"Vinegar Available" )
      Coil( #Vinegar_EN )
   END_RUNG
   // the same network as SCL:
   #Vinegar_EN := #alwaysON AND #State."Dose EN" AND #"Vinegar Available";
END_REGION

REGION Network 32: Vinegar Setpoint
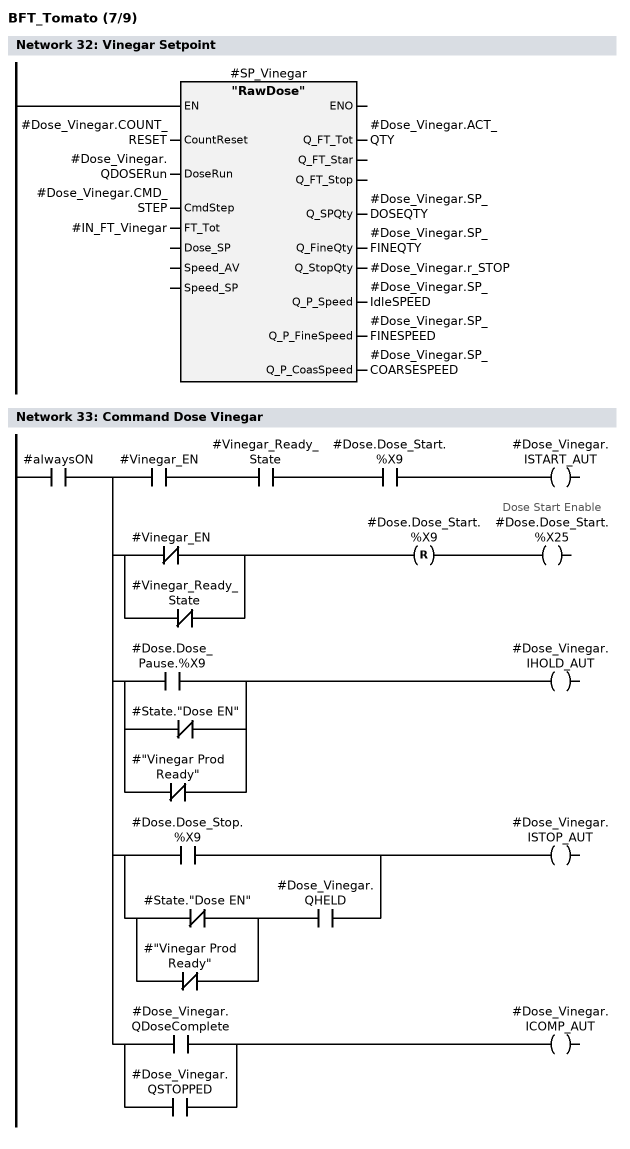
   RUNG wire#powerrail
      #SP_Vinegar(CountReset := #Dose_Vinegar.COUNT_RESET, DoseRun := #Dose_Vinegar.QDOSERun, CmdStep := #Dose_Vinegar.CMD_STEP, FT_Tot := #IN_FT_Vinegar, Dose_SP :=, Speed_AV :=, Speed_SP :=, Q_FT_Tot => #Dose_Vinegar.ACT_QTY, Q_FT_Star =>, Q_FT_Stop =>, Q_SPQty => #Dose_Vinegar.SP_DOSEQTY, Q_FineQty => #Dose_Vinegar.SP_FINEQTY, Q_StopQty => #Dose_Vinegar.r_STOP, Q_P_Speed => #Dose_Vinegar.SP_IdleSPEED, Q_P_FineSpeed => #Dose_Vinegar.SP_FINESPEED, Q_P_CoasSpeed => #Dose_Vinegar.SP_COARSESPEED)
   END_RUNG
   // the same network as SCL:
   #SP_Vinegar(CountReset := #Dose_Vinegar.COUNT_RESET,   // "RawDose"
               DoseRun := #Dose_Vinegar.QDOSERun,
               CmdStep := #Dose_Vinegar.CMD_STEP,
               FT_Tot := #IN_FT_Vinegar,
               Q_FT_Tot => #Dose_Vinegar.ACT_QTY,
               Q_SPQty => #Dose_Vinegar.SP_DOSEQTY,
               Q_FineQty => #Dose_Vinegar.SP_FINEQTY,
               Q_StopQty => #Dose_Vinegar.r_STOP,
               Q_P_Speed => #Dose_Vinegar.SP_IdleSPEED,
               Q_P_FineSpeed => #Dose_Vinegar.SP_FINESPEED,
               Q_P_CoasSpeed => #Dose_Vinegar.SP_COARSESPEED);
END_REGION

REGION Network 33: Command Dose Vinegar
   RUNG wire#powerrail
      Contact( #alwaysON )
      wire#w1
      Contact( #Vinegar_EN )
      Contact( #Vinegar_Ready_State )
      Contact( #Dose.Dose_Start.%X9 )
      Coil( #Dose_Vinegar.ISTART_AUT )
   END_RUNG
   RUNG wire#w1
      I_Contact( #Vinegar_EN )
      wire#w2
      R_Coil( #Dose.Dose_Start.%X9 )
      Coil( #Dose.Dose_Start.%X25 )   // Dose Start Enable
   END_RUNG
   RUNG wire#w1
      I_Contact( #Vinegar_Ready_State )
   END_RUNG wire#w2
   RUNG wire#w1
      Contact( #Dose.Dose_Pause.%X9 )
      wire#w3
      Coil( #Dose_Vinegar.IHOLD_AUT )
   END_RUNG
   RUNG wire#w1
      I_Contact( #State."Dose EN" )
   END_RUNG wire#w3
   RUNG wire#w1
      I_Contact( #"Vinegar Prod Ready" )
   END_RUNG wire#w3
   RUNG wire#w1
      Contact( #Dose.Dose_Stop.%X9 )
      wire#w4
      Coil( #Dose_Vinegar.ISTOP_AUT )
   END_RUNG
   RUNG wire#w1
      I_Contact( #State."Dose EN" )
      wire#w5
      Contact( #Dose_Vinegar.QHELD )
   END_RUNG wire#w4
   RUNG wire#w1
      I_Contact( #"Vinegar Prod Ready" )
   END_RUNG wire#w5
   RUNG wire#w1
      Contact( #Dose_Vinegar.QDoseComplete )
      wire#w6
      Coil( #Dose_Vinegar.ICOMP_AUT )
   END_RUNG
   RUNG wire#w1
      Contact( #Dose_Vinegar.QSTOPPED )
   END_RUNG wire#w6
   // the same network as SCL:
   #Dose_Vinegar.ISTART_AUT := #alwaysON AND #Vinegar_EN AND #Vinegar_Ready_State AND #Dose.Dose_Start.%X9;
   #_w1 := #alwaysON AND (NOT #Vinegar_EN OR NOT #Vinegar_Ready_State);
   IF #_w1 THEN #Dose.Dose_Start.%X9 := FALSE; END_IF;
   #Dose.Dose_Start.%X25 := #_w1;   // Dose Start Enable
   #Dose_Vinegar.IHOLD_AUT := #alwaysON AND (#Dose.Dose_Pause.%X9 OR NOT #State."Dose EN" OR NOT #"Vinegar Prod Ready");
   #Dose_Vinegar.ISTOP_AUT := #alwaysON AND (#Dose.Dose_Stop.%X9 OR ((NOT #State."Dose EN" OR NOT #"Vinegar Prod Ready") AND #Dose_Vinegar.QHELD));
   #Dose_Vinegar.ICOMP_AUT := #alwaysON AND (#Dose_Vinegar.QDoseComplete OR #Dose_Vinegar.QSTOPPED);
END_REGION

REGION Network 34: Dose Vinegar
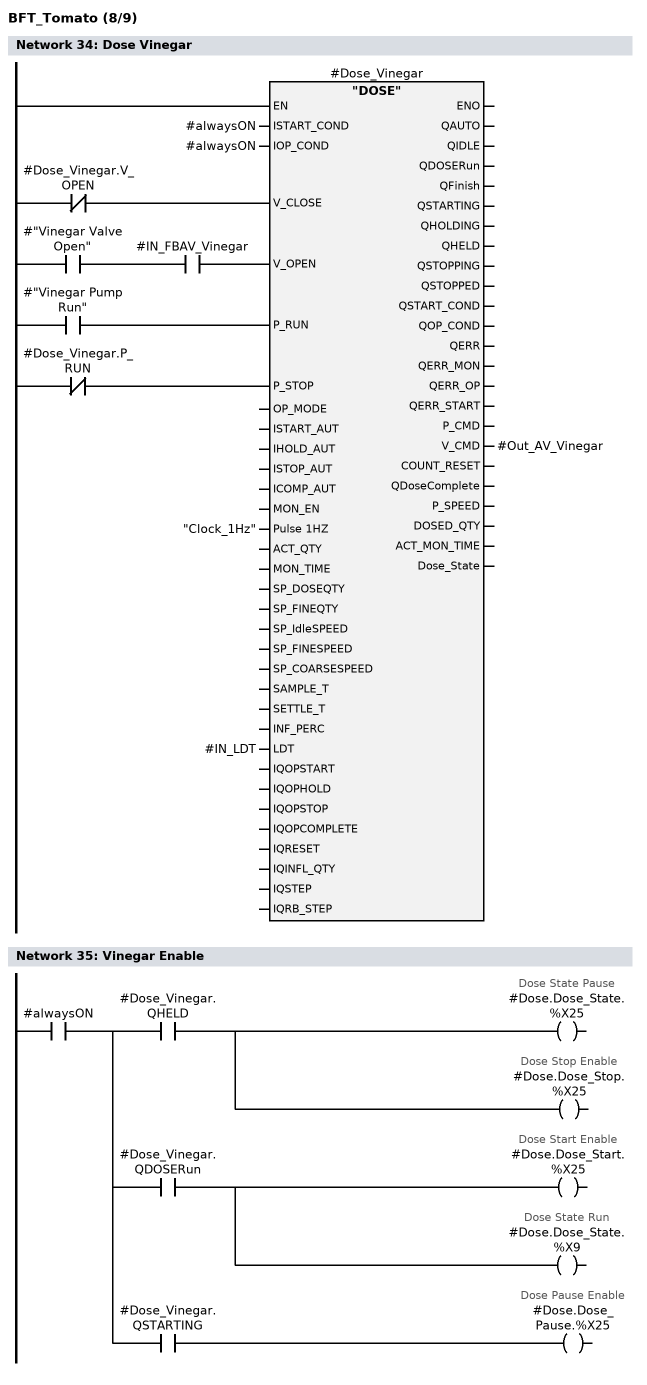
   RUNG wire#powerrail
      #Dose_Vinegar(V_CLOSE := wire#w1, V_OPEN := wire#w2, P_RUN := wire#w3, P_STOP := wire#w4, ISTART_COND := #alwaysON, IOP_COND := #alwaysON, OP_MODE :=, ISTART_AUT :=, IHOLD_AUT :=, ISTOP_AUT :=, ICOMP_AUT :=, MON_EN :=, "Pulse 1HZ" := "Clock_1Hz", ACT_QTY :=, MON_TIME :=, SP_DOSEQTY :=, SP_FINEQTY :=, SP_IdleSPEED :=, SP_FINESPEED :=, SP_COARSESPEED :=, SAMPLE_T :=, SETTLE_T :=, INF_PERC :=, LDT := #IN_LDT, IQOPSTART :=, IQOPHOLD :=, IQOPSTOP :=, IQOPCOMPLETE :=, IQRESET :=, IQINFL_QTY :=, IQSTEP :=, IQRB_STEP :=, QAUTO =>, QIDLE =>, QDOSERun =>, QFinish =>, QSTARTING =>, QHOLDING =>, QHELD =>, QSTOPPING =>, QSTOPPED =>, QSTART_COND =>, QOP_COND =>, QERR =>, QERR_MON =>, QERR_OP =>, QERR_START =>, P_CMD =>, V_CMD => #Out_AV_Vinegar, COUNT_RESET =>, QDoseComplete =>, P_SPEED =>, DOSED_QTY =>, ACT_MON_TIME =>, Dose_State =>)
   END_RUNG
   RUNG wire#powerrail
      I_Contact( #Dose_Vinegar.V_OPEN )
   END_RUNG wire#w1
   RUNG wire#powerrail
      Contact( #"Vinegar Valve Open" )
      Contact( #IN_FBAV_Vinegar )
   END_RUNG wire#w2
   RUNG wire#powerrail
      Contact( #"Vinegar Pump Run" )
   END_RUNG wire#w3
   RUNG wire#powerrail
      I_Contact( #Dose_Vinegar.P_RUN )
   END_RUNG wire#w4
   // the same network as SCL:
   #Dose_Vinegar(ISTART_COND := #alwaysON,   // "DOSE"
                 IOP_COND := #alwaysON,
                 V_CLOSE := NOT #Dose_Vinegar.V_OPEN,
                 V_OPEN := #"Vinegar Valve Open" AND #IN_FBAV_Vinegar,
                 P_RUN := #"Vinegar Pump Run",
                 P_STOP := NOT #Dose_Vinegar.P_RUN,
                 "Pulse 1HZ" := "Clock_1Hz",
                 LDT := #IN_LDT,
                 V_CMD => #Out_AV_Vinegar);
END_REGION

REGION Network 35: Vinegar Enable
   RUNG wire#powerrail
      Contact( #alwaysON )
      wire#w1
      Contact( #Dose_Vinegar.QHELD )
      wire#w2
      Coil( #Dose.Dose_State.%X25 )   // Dose State Pause
   END_RUNG
   RUNG wire#w2
      Coil( #Dose.Dose_Stop.%X25 )   // Dose Stop Enable
   END_RUNG
   RUNG wire#w1
      Contact( #Dose_Vinegar.QDOSERun )
      wire#w3
      Coil( #Dose.Dose_Start.%X25 )   // Dose Start Enable
   END_RUNG
   RUNG wire#w3
      Coil( #Dose.Dose_State.%X9 )   // Dose State Run
   END_RUNG
   RUNG wire#w1
      Contact( #Dose_Vinegar.QSTARTING )
      Coil( #Dose.Dose_Pause.%X25 )   // Dose Pause Enable
   END_RUNG
   // the same network as SCL:
   #Dose.Dose_State.%X25 := #alwaysON AND #Dose_Vinegar.QHELD;   // Dose State Pause
   #Dose.Dose_Stop.%X25 := #Dose.Dose_State.%X25;   // Dose Stop Enable
   #Dose.Dose_Start.%X25 := #alwaysON AND #Dose_Vinegar.QDOSERun;   // Dose Start Enable
   #Dose.Dose_State.%X9 := #Dose.Dose_Start.%X25;   // Dose State Run
   #Dose.Dose_Pause.%X25 := #alwaysON AND #Dose_Vinegar.QSTARTING;   // Dose Pause Enable
END_REGION

REGION Network 36: Vinegar Header Req
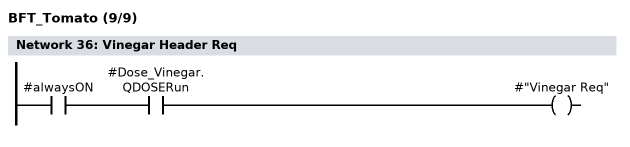
   RUNG wire#powerrail
      Contact( #alwaysON )
      Contact( #Dose_Vinegar.QDOSERun )
      Coil( #"Vinegar Req" )
   END_RUNG
   // the same network as SCL:
   #"Vinegar Req" := #alwaysON AND #Dose_Vinegar.QDOSERun;
END_REGION
END_FUNCTION_BLOCK
